PROGRAM P_Demo_FB_DMXClearStatusId
VAR
    fbClearStatus     : FB_DMXClearStatusId;          // 清设备消息缓冲
    stDmxCmdBuffer    : ST_DMXCommandBuffer;          // 与通讯 FB 共用
    wTargetManufId    : WORD := 16#4241;              // 目标灯具厂商 ID
    dwTargetDeviceId  : DWORD := 16#12131415;         // 目标灯具设备 ID
    byTargetPort      : BYTE := 0;                    // 根设备通道 0
    bDoClear          : BOOL := FALSE;                // 在线给一次上升沿触发
    bBusy             : BOOL;
    bError            : BOOL;
    udiErrId          : UDINT;
END_VAR

// ============================================================
// Tc2_DMX.FB_DMXClearStatusId 演示程序
// ============================================================
// 场景：故障处理闭环：PLC 读出某灯状态消息并上报后，确认处理完毕清掉该灯消息缓冲。
// 价值：把设备消息缓冲清除做成 PLC 调用，实现读-处理-清的标准故障闭环，避免重复报警。
// 验证：先用 FB_DMXGetStatusMessages 确认有消息，给 bDoClear 一次上升沿 -> bBusy 短暂 TRUE -> 回 FALSE 后再读 FB_DMXGetStatusMessages 应不再返回已清消息。
// 验证步骤：
//   1. 右键 PLC 项目下 POUs 文件夹 → Add → Existing Item → 选本 .TcPOU 文件
//   2. 引用 Tc2_DMX；同项目里放一个 FB_EL6851CommunicationEx 实例并共用 stDmxCmdBuffer（非 CycleMode）
//   3. 编译 → 登录 → 运行；按上方『验证』行在线给上升沿观察
// ============================================================

fbClearStatus(
    bStart                     := bDoClear,
    wDestinationManufacturerId := wTargetManufId,
    dwDestinationDeviceId      := dwTargetDeviceId,
    byPortId                   := byTargetPort,
    dwOptions                  := 0,
    stCommandBuffer            := stDmxCmdBuffer,
    bBusy                      => bBusy,
    bError                     => bError,
    udiErrorId                 => udiErrId
);

END_PROGRAM

(* stored: Version 1.1.0.1, ProductVersion 3.1.4024.5
   POU P_Demo_FB_DMXClearStatusId: Id {64386ca4-84b2-5199-825c-1d1f4eefe324}, SpecialFunc None *)
